// TIA Portal V16 export
// export: Created 2021-04-06T19:52:15.0270381Z, ExportSetting WithDefaults, DisplayName Totally Integrated Automation Portal, DisplayVersion V16, DisplayName TIA Portal Version Control Interface, DisplayVersion V16, DisplayName TIA Portal Openness, DisplayVersion V16, DisplayName STEP 7 Professional, DisplayVersion V16, DisplayName STEP 7 Safety, DisplayVersion V16, DisplayName WinCC Unified SCADA Engineering System, DisplayVersion V16
FUNCTION_BLOCK "modbus_FB"   // FB9, LAD
{ S7_Optimized_Access := 'TRUE' }
VERSION : 0.1
// stored: AutoNumber true, IsIECCheckEnabled false, IsRetainMemResEnabled false, MemoryReserve 100, SetENOAutomatically false, UDAEnableTagReadback false
   VAR_IN_OUT
      currentWeight : Array[0..12] of Real;
   END_VAR
   VAR
      MODBUS_ADDRESS : Array[0..12] of UInt;
      modbus_SenecaConnectPort1_FB { S7_SetPoint := 'True'} : "modbus_SenecaConnectPort1";
      modbus_SenecaConnectPort2_FB { S7_SetPoint := 'True'} : "modbus_SenecaConnectPort2";
   END_VAR
   VAR_TEMP
      i : SInt;
   END_VAR
   // MODBUS_ADDRESS[1] := 10;
   // MODBUS_ADDRESS[2] := 11;
   // MODBUS_ADDRESS[3] := 12;
   // MODBUS_ADDRESS[4] := 13;
   // MODBUS_ADDRESS[5] := 14;
   // MODBUS_ADDRESS[6] := 15;
   // MODBUS_ADDRESS[7] := 20;
   // MODBUS_ADDRESS[8] := 21;
   // MODBUS_ADDRESS[9] := 22;
   // MODBUS_ADDRESS[10] := 23;
   // MODBUS_ADDRESS[11] := 24;
   // MODBUS_ADDRESS[12] := 25;
BEGIN

REGION Network 1: ОПРОС МОДУЛЕЙ ЧЕРЕРЗ 1 ПОРТ
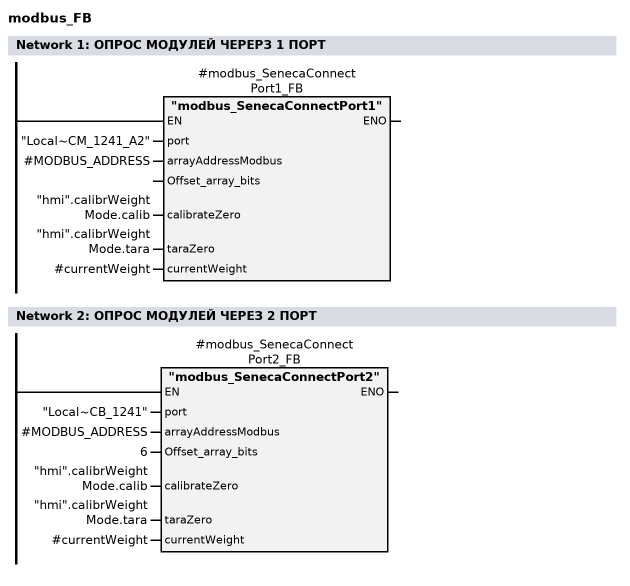
   RUNG wire#powerrail
      #modbus_SenecaConnectPort1_FB(port := "Local~CM_1241_A2", arrayAddressModbus := #MODBUS_ADDRESS, Offset_array_bits :=, calibrateZero := "hmi".calibrWeightMode.calib, taraZero := "hmi".calibrWeightMode.tara, currentWeight := #currentWeight)
   END_RUNG
   // the same network as SCL:
   #modbus_SenecaConnectPort1_FB(port := "Local~CM_1241_A2",   // "modbus_SenecaConnectPort1"
                           arrayAddressModbus := #MODBUS_ADDRESS,
                           calibrateZero := "hmi".calibrWeightMode.calib,
                           taraZero := "hmi".calibrWeightMode.tara,
                           currentWeight := #currentWeight);
END_REGION

REGION Network 2: ОПРОС МОДУЛЕЙ ЧЕРЕЗ 2 ПОРТ
   RUNG wire#powerrail
      #modbus_SenecaConnectPort2_FB(port := "Local~CB_1241", arrayAddressModbus := #MODBUS_ADDRESS, Offset_array_bits := 6, calibrateZero := "hmi".calibrWeightMode.calib, taraZero := "hmi".calibrWeightMode.tara, currentWeight := #currentWeight)
   END_RUNG
   // the same network as SCL:
   #modbus_SenecaConnectPort2_FB(port := "Local~CB_1241",   // "modbus_SenecaConnectPort2"
                           arrayAddressModbus := #MODBUS_ADDRESS,
                           Offset_array_bits := 6,
                           calibrateZero := "hmi".calibrWeightMode.calib,
                           taraZero := "hmi".calibrWeightMode.tara,
                           currentWeight := #currentWeight);
END_REGION

REGION Network 3 (SCL): Передаем вес в панель
   #i := 0;
   FOR #i := 1 TO 12 DO
       "hmi".weightLine[#i].currentWeightPocket := #currentWeight[#i];
   END_FOR;
END_REGION

REGION Network 4 (SCL)
   IF "hmi".calibrWeightMode.tara[0] THEN
       #i := 0;
       FOR #i := 1 TO 12 DO
           "hmi".calibrWeightMode.tara[#i] := true;
       END_FOR;
   END_IF;
END_REGION
END_FUNCTION_BLOCK
